Fanuc KAREL source: NC0070.KL

-- PROVISIONAL review KL for V1013-1; original PC SHA256 df03d81601bfb2832907b86c3830f55604e0f6083c8fb011b607eeeccf8fd210
-- Incomplete behavior may be omitted. Consult companion uncertainty JSON. Do not deploy.
PROGRAM NC0070
%NOLOCKGROUP
-- UNRESOLVED_LOCAL_POOL 19 cells at code offset 3; source declarations unknown
-- DIRECT_LOCAL_WORD_ACCESS alone does not prove INTEGER, REAL, or BOOLEAN
BEGIN
  -- UNRESOLVED_PC offsets 0-8; opcodes 2B,2C,7B
  -- UNRESOLVED_PC offsets 13-20; opcodes 9D,23
  -- UNRESOLVED_PC offsets 25-54; opcodes 9D,23,9E,2E,22,7A
  -- UNRESOLVED_PC offsets 59-88; opcodes 9D,23,9E,2E,22,7A
  -- UNRESOLVED_PC offsets 93-122; opcodes 9D,23,9E,2E,22,7A
  -- UNRESOLVED_PC offsets 127-156; opcodes 9D,23,9E,2E,22,7A
  -- UNRESOLVED_PC offsets 161-190; opcodes 9D,23,9E,2E,22,7A
  -- UNRESOLVED_PC offsets 195-224; opcodes 9D,23,9E,2E,22,7A
  -- UNRESOLVED_PC offsets 229-258; opcodes 9D,23,9E,2E,22,7A
  -- UNRESOLVED_PC offsets 263-292; opcodes 9D,23,9E,2E,22,7A
  -- UNRESOLVED_PC offsets 297-326; opcodes 9D,23,9E,2E,22,7A
  -- UNRESOLVED_PC offsets 331-360; opcodes 9D,23,9E,2E,22,7A
  -- UNRESOLVED_PC offsets 365-394; opcodes 9D,23,9E,2E,22,7A
  -- UNRESOLVED_PC offsets 399-428; opcodes 9D,23,9E,2E,22,7A
  -- UNRESOLVED_PC offsets 433-462; opcodes 9D,23,9E,2E,22,7A
  -- UNRESOLVED_PC offsets 467-496; opcodes 9D,23,9E,2E,22,7A
  -- UNRESOLVED_PC offsets 501-530; opcodes 9D,23,9E,2E,22,7A
  -- UNRESOLVED_PC offsets 535-564; opcodes 9D,23,9E,2E,22,7A
  -- UNRESOLVED_PC offsets 569-598; opcodes 9D,23,9E,2E,22,7A
  -- UNRESOLVED_PC offsets 603-632; opcodes 9D,23,9E,2E,22,7A
  -- UNRESOLVED_PC offsets 637-651; opcodes 21,9D,52,23
  -- UNRESOLVED_PC offsets 656-671; opcodes 20,2C,23
  -- UNRESOLVED_PC offsets 676-691; opcodes 20,2C,23
  -- UNRESOLVED_PC offsets 696-711; opcodes 20,2C,23
  -- UNRESOLVED_PC offsets 716-731; opcodes 20,2C,23
  -- UNRESOLVED_PC offsets 736-751; opcodes 20,2C,23
  -- UNRESOLVED_PC offsets 756-771; opcodes 20,2C,23
  -- UNRESOLVED_PC offsets 776-791; opcodes 20,2C,23
  -- UNRESOLVED_PC offsets 796-811; opcodes 20,2C,23
  -- UNRESOLVED_PC offsets 816-831; opcodes 20,2C,23
  -- UNRESOLVED_PC offsets 836-851; opcodes 20,2C,23
  -- UNRESOLVED_PC offsets 856-871; opcodes 20,2C,23
  -- UNRESOLVED_PC offsets 876-891; opcodes 20,2C,23
  -- UNRESOLVED_PC offsets 896-911; opcodes 20,2C,23
  -- UNRESOLVED_PC offsets 916-931; opcodes 20,2C,23
  -- UNRESOLVED_PC offsets 936-951; opcodes 20,2C,23
  -- UNRESOLVED_PC offsets 956-971; opcodes 20,2C,23
  -- UNRESOLVED_PC offsets 976-991; opcodes 20,2C,23
  -- UNRESOLVED_PC offsets 996-1011; opcodes 20,2C,23
  -- UNRESOLVED_PC offsets 1016-1020; opcodes 7F
  -- UNRESOLVED_PC offsets 1025-1029; opcodes 27,AA
  -- UNRESOLVED_PC offsets 1034-1038; opcodes 7F
END NC0070
